FUNCTION_BLOCK Composite1
  (* Standard: 61499-2 *)
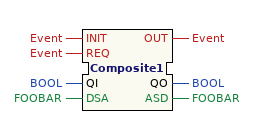
  EVENT_INPUT
    INIT;
    REQ;
  END_EVENT
  EVENT_OUTPUT
    OUT;
  END_EVENT
  VAR_INPUT
    QI : BOOL;
  END_VAR
  VAR_OUTPUT
    QO : BOOL;
  END_VAR
  SOCKETS
    DSA : FOOBAR;
  END_SOCKETS
  PLUGS
    ASD : FOOBAR;
  END_PLUGS
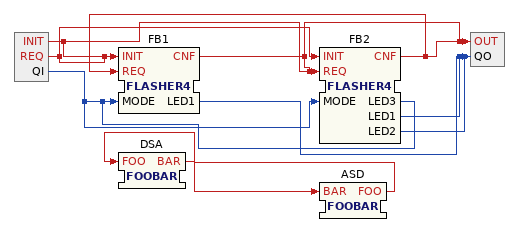
  FBS
    FB1 : FLASHER4;
    FB2 : FLASHER4;
  END_FBS
  EVENT_CONNECTIONS
    INIT TO FB1.INIT;
    REQ TO FB1.INIT;
    FB2.CNF TO FB1.REQ;
    FB2.CNF TO OUT;
    REQ TO FB2.INIT;
    FB1.CNF TO OUT;
    INIT TO FB2.REQ;
    ASD.FOO TO DSA.FOO;
    DSA.BAR TO ASD.BAR;
    FB1.CNF TO FB2.REQ;
  END_CONNECTIONS
  DATA_CONNECTIONS
    FB2.LED3 TO FB1.MODE;
    QI TO FB1.MODE;
    FB1.LED1 TO QO;
    QI TO FB2.MODE;
    FB2.LED1 TO QO;
    FB2.LED2 TO QO;
  END_CONNECTIONS
END_FUNCTION_BLOCK
